// TIA Portal V20 export
// export: Created 2026-04-11T06:02:30.045527Z, ExportSetting WithDefaults, DisplayName Totally Integrated Automation Portal, DisplayVersion V20, DisplayName TIA Portal Openness, DisplayVersion V20, DisplayName TIA Portal Version Control Interface, DisplayVersion V20, DisplayName STEP 7 Professional, DisplayVersion V20, DisplayName STEP 7 Safety, DisplayVersion V20, DisplayName WinCC Basic/Comfort/Advanced, DisplayVersion V20, DisplayName WinCC Unified, DisplayVersion V20
TYPE "udtError_SiwarexU"
// stored: IsFailsafeCompliant false
   STRUCT
      GroupError { ExternalWritable := 'False'} : Bool;   // Grpoup error, check module
      WriteAccessFailed { ExternalWritable := 'False'} : Bool;   // Module write access error
      CalibrationNeeded { ExternalWritable := 'False'} : Bool;   // Scale not adjusted, need calibration
      UpdateTimeout { ExternalWritable := 'False'} : Bool;   // Module update time out
   END_STRUCT;
END_TYPE
